Omron CX-Programmer project NewProject (CX-Programmer 9.20)

# PLC PBL: CP1E NA

## Global symbols (name address type ; comment)
0.00 BOOL  ; START
0.01 BOOL  ; STOP
0.02 BOOL  ; BOTTEL SENSOR
0.03 BOOL  ; CAPPING S
0.04 BOOL  ; PACKED BOTTEL
0.05 BOOL  ; REST
0.06 BOOL  ; PACKING S
0.08 BOOL  ; rest
0.10 BOOL  ; do
100.00 BOOL  ; CONVEYOR
100.01 BOOL  ; FILLING BARRIER
100.02 BOOL  ; FILLING VALVE
100.03 BOOL  ; CAPPING BARRIER
100.04 BOOL  ; CAPPING
100.05 BOOL  ; Filling Motor
100.06 BOOL  ; BACKING CYLINDER
100.07 BOOL  ; PACKING CONVEYOR
C000 BOOL  ; conter
C006 BOOL  ; BOTTEL COUNTER
T000 BOOL  ; Sauce container
T001 BOOL  ; TIMER
T002 BOOL  ; TIMER2
T003 BOOL  ; DELAY
T004 BOOL  ; DELAY2
T005 BOOL  ; Filling timer

## Program NewProgram1 (cyclic task 0)

### Section Section1

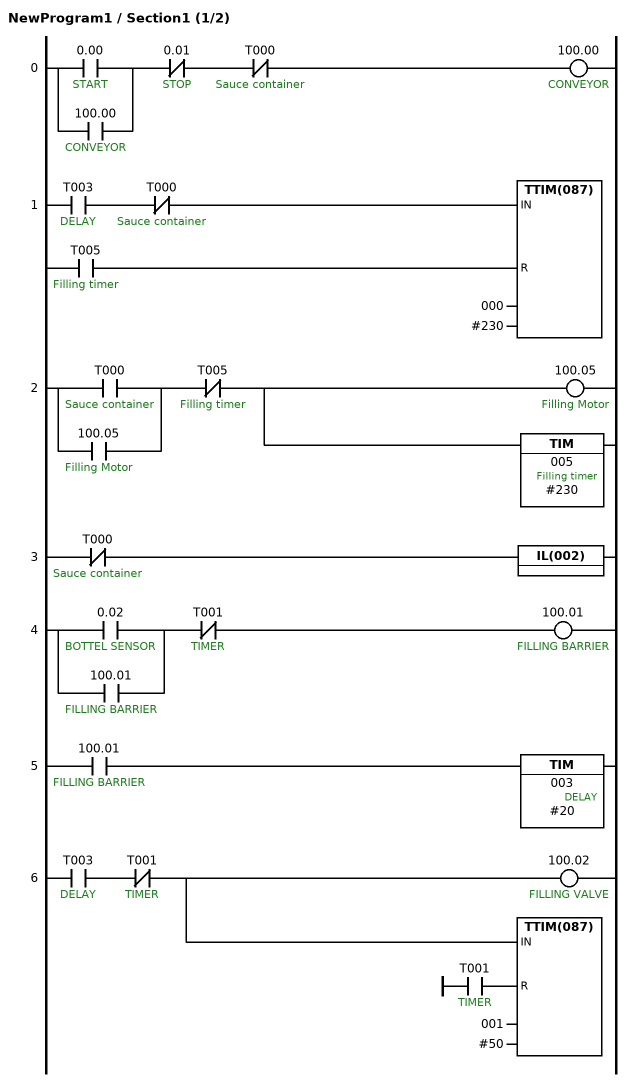
; rung 0
LD 0.00  ; START
OR 100.00  ; CONVEYOR
ANDNOT 0.01  ; STOP
ANDNOT T000  ; Sauce container
OUT 100.00  ; CONVEYOR
; rung 1
LD T003  ; DELAY
ANDNOT T000  ; Sauce container
LD T005  ; Filling timer
TTIM(087) 000 #230  ; Sauce container
; rung 2
LD T000  ; Sauce container
OR 100.05  ; Filling Motor
ANDNOT T005  ; Filling timer
OUT 100.05  ; Filling Motor
TIM 005 #230  ; Filling timer
; rung 3
LDNOT T000  ; Sauce container
IL(002)
; rung 4
LD 0.02  ; BOTTEL SENSOR
OR 100.01  ; FILLING BARRIER
ANDNOT T001  ; TIMER
OUT 100.01  ; FILLING BARRIER
; rung 5
LD 100.01  ; FILLING BARRIER
TIM 003 #20  ; DELAY
; rung 6
LD T003  ; DELAY
ANDNOT T001  ; TIMER
OUT 100.02  ; FILLING VALVE
LD T001  ; TIMER
TTIM(087) 001 #50  ; TIMER

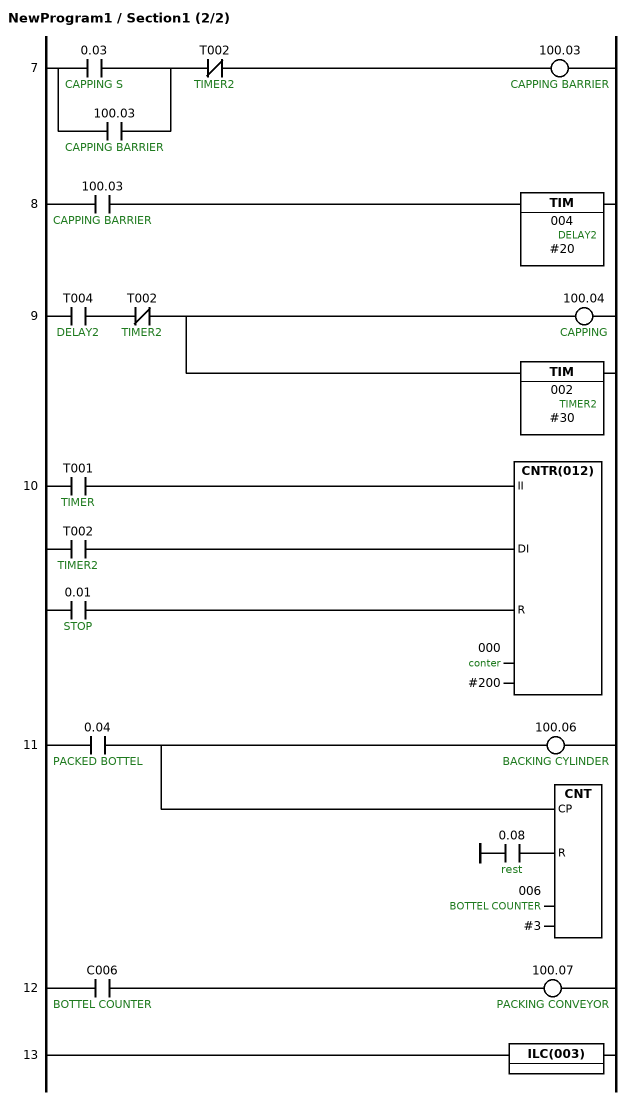
; rung 7
LD 0.03  ; CAPPING S
OR 100.03  ; CAPPING BARRIER
ANDNOT T002  ; TIMER2
OUT 100.03  ; CAPPING BARRIER
; rung 8
LD 100.03  ; CAPPING BARRIER
TIM 004 #20  ; DELAY2
; rung 9
LD T004  ; DELAY2
ANDNOT T002  ; TIMER2
OUT 100.04  ; CAPPING
TIM 002 #30  ; TIMER2
; rung 10
LD T001  ; TIMER
LD T002  ; TIMER2
LD 0.01  ; STOP
CNTR(012) 000 #200  ; conter
; rung 11
LD 0.04  ; PACKED BOTTEL
OUT 100.06  ; BACKING CYLINDER
LD 0.08  ; rest
CNT 006 #3  ; BOTTEL COUNTER
; rung 12
LD C006  ; BOTTEL COUNTER
OUT 100.07  ; PACKING CONVEYOR
; rung 13
ILC(003)

### Section END
; rung 0
END(001)